{attribute 'qualified_only'}
{attribute 'strict'}
TYPE SafetyStatus :
(
	UNKNOWN := 0,
	READY	:=1,
	SAFETY_STOPPED	:=2,
	ERROR	:=3	
);
END_TYPE

(* stored: Version 1.1.0.1, ProductVersion 3.1.4024.12
   DUT SafetyStatus: Id {d0420daa-9c74-458e-98b3-20475ec7832d} *)
